FUNCTION_BLOCK CAT_Conveyor_1 (* Composite Function Block Type *)
  (* Standard: 61499-2 *)
  (* Version 0.0, 16/08/2021, prana, nxtControl GmBH, template *)
  PACKAGE Main;
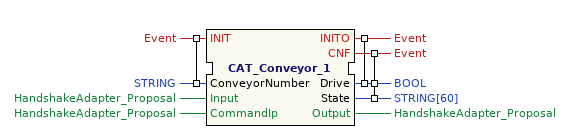
  EVENT_INPUT
    INIT WITH ConveyorNumber; (* Initialization Request *)
  END_EVENT
  EVENT_OUTPUT
    INITO WITH Drive; (* Initialization Confirm *)
    CNF WITH Drive, State; (* Execution Confirmation *)
  END_EVENT
  VAR_INPUT
    ConveyorNumber : STRING;
  END_VAR
  VAR_OUTPUT
    Drive : BOOL; (* Output event qualifier *)
    State : STRING[60];
  END_VAR
  SOCKETS
    Input : HandshakeAdapter_Proposal;
    CommandIp : HandshakeAdapter_Proposal;
  END_SOCKETS
  PLUGS
    Output : HandshakeAdapter_Proposal;
  END_PLUGS
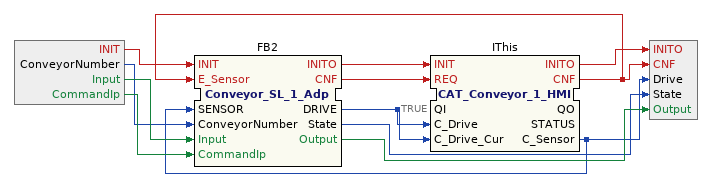
  FBS
    IThis : CAT_Conveyor_1_HMI(QI := TRUE);
    FB2 : Conveyor_SL_1_Adp;
  END_FBS
  EVENT_CONNECTIONS
    INIT TO FB2.INIT;
    FB2.INITO TO IThis.INIT;
    FB2.CNF TO IThis.REQ;
    IThis.INITO TO INITO;
    IThis.CNF TO FB2.E_Sensor;
    IThis.CNF TO CNF;
  END_CONNECTIONS
  DATA_CONNECTIONS
    FB2.DRIVE TO IThis.C_Drive;
    FB2.DRIVE TO IThis.C_Drive_Cur;
    IThis.C_Sensor TO FB2.SENSOR;
    IThis.C_Sensor TO Drive;
    ConveyorNumber TO FB2.ConveyorNumber;
    FB2.State TO State;
  END_CONNECTIONS
  ADAPTER_CONNECTIONS
    Input TO FB2.Input;
    FB2.Output TO Output;
    CommandIp TO FB2.CommandIp;
  END_CONNECTIONS
END_FUNCTION_BLOCK
